Staubli VAL3: S2S_demo_0.pjx

--- S2S_demo_0.pjx ---
Parameters version=s7.9.1 stackSize=5000 millimeterUnit=true
Program file=start.pgx
Program file=stop.pgx
Data file=S2S_demo_0.dtx
Library alias=S7 path=Disk://S2S/S2S.pjx

--- S2S_demo_0.dtx ---
sio sTcpClient = {link=Socket\sTcpClient}
num nDBnumber = 1
num nDB[100]
  [0] = 1
  [1] = 2
  [2] = 3
  [3] = 4
  [4] = 5
  [5] = 6
  [6] = 7
  [7] = 8
  [8] = 9
  [9] = 10
  [10] = 1
  [11] = 2
  [12] = 3
  [13] = 4
  [14] = 5
  [15] = 6
  [16] = 7
  [17] = 8
  [18] = 9
  [19] = 10
  [20] = 1
  [21] = 2
  [22] = 3
  [23] = 4
  [24] = 5
  [25] = 6
  [26] = 7
  [27] = 8
  [28] = 9
  [29] = 10
  [30] = 1
  [31] = 2
  [32] = 3
  [33] = 4
  [34] = 5
  [35] = 6
  [36] = 7
  [37] = 8
  [38] = 9
  [39] = 10
  [40] = 1
  [41] = 2
  [42] = 3
  [43] = 4
  [44] = 5
  [45] = 6
  [46] = 7
  [47] = 8
  [48] = 9
  [49] = 10
  [50] = 1
  [51] = 2
  [52] = 3
  [53] = 4
  [54] = 5
  [55] = 6
  [56] = 7
  [57] = 8
  [58] = 9
  [59] = 10
  [60] = 1
  [61] = 2
  [62] = 3
  [63] = 4
  [64] = 5
  [65] = 6
  [66] = 7
  [67] = 8
  [68] = 9
  [69] = 10
  [70] = 1
  [71] = 2
  [72] = 3
  [73] = 4
  [74] = 5
  [75] = 6
  [76] = 7
  [77] = 8
  [78] = 9
  [79] = 10
  [80] = 1
  [81] = 2
  [82] = 3
  [83] = 4
  [84] = 5
  [85] = 6
  [86] = 7
  [87] = 8
  [88] = 9
  [89] = 10
  [90] = 1
  [91] = 2
  [92] = 3
  [93] = 4
  [94] = 5
  [95] = 6
  [96] = 7
  [97] = 8
  [98] = 9
  [99] = 10
num nSampleBuffer[300]
  [0] = 1
  [1] = 211
  [2] = 3
  [3] = 4
  [4] = 5
  [5] = 6
  [6] = 7
  [7] = 8
  [8] = 9
  [9] = 10
  [10] = 1
  [11] = 2
  [12] = 3
  [13] = 4
  [14] = 5
  [15] = 6
  [16] = 7
  [17] = 8
  [18] = 9
  [19] = 10
  [20] = 1
  [21] = 2
  [22] = 3
  [23] = 4
  [24] = 5
  [25] = 6
  [26] = 7
  [27] = 8
  [28] = 9
  [29] = 10
  [30] = 1
  [31] = 2
  [32] = 3
  [33] = 4
  [34] = 5
  [35] = 6
  [36] = 7
  [37] = 8
  [38] = 9
  [39] = 10
  [40] = 1
  [41] = 2
  [42] = 3
  [43] = 4
  [44] = 5
  [45] = 6
  [46] = 7
  [47] = 8
  [48] = 9
  [49] = 10
  [50] = 1
  [51] = 2
  [52] = 3
  [53] = 4
  [54] = 5
  [55] = 6
  [56] = 7
  [57] = 8
  [58] = 9
  [59] = 10
  [60] = 1
  [61] = 2
  [62] = 3
  [63] = 4
  [64] = 5
  [65] = 6
  [66] = 7
  [67] = 8
  [68] = 9
  [69] = 10
  [70] = 1
  [71] = 2
  [72] = 3
  [73] = 4
  [74] = 5
  [75] = 6
  [76] = 7
  [77] = 8
  [78] = 9
  [79] = 10
  [80] = 1
  [81] = 2
  [82] = 3
  [83] = 4
  [84] = 5
  [85] = 6
  [86] = 7
  [87] = 8
  [88] = 9
  [89] = 10
  [90] = 1
  [91] = 2
  [92] = 3
  [93] = 4
  [94] = 5
  [95] = 6
  [96] = 7
  [97] = 8
  [98] = 9
  [99] = 10
  [236] = 5
  [237] = 7
  [238] = 6
  [253] = 77
  [254] = 6
  [255] = 5
  [266] = 33
  [281] = 31
  [299] = 99
num nTimer

--- stop.pgx ---
program stop()
begin
end
